TYPE DUT_RecipeCommand :
STRUCT
	SkillID: INT;
	SkillName: STRING(80);
	Quantity: LREAL;
END_STRUCT
END_TYPE

(* stored: Version 1.1.0.1, ProductVersion 3.1.0.25
   DUT DUT_RecipeCommand: Id {52c460f9-1dcf-4ec9-a724-38e053a613ed} *)
